// TwinCAT 3 PLC project plc_lfe_vac_fs
// ProgramVersion: 3.1.4022.7
// libraries:
//   L2SI Vacuum Library, * (SLAC)
//   LCLS General, * (SLAC)
//   PMPS, * (SLAC - LCLS)
//   Tc2_Standard, * (Beckhoff Automation GmbH)
//   Tc2_System, * (Beckhoff Automation GmbH)
//   Tc3_Module, * (Beckhoff Automation GmbH)
// project tree:
//   GVLs/ GVL_FS_Devices.TcGVL (not stored)
//   / PlcTask.TcTTO
//   POUs/ MAIN_FS.TcPOU
// (motion and I/O tree: see PLC project plc_lfe_vac)
// real-time tasks:
//   TASK PlcTask: cycle T#10ms, priority 20, ADS port 350
// variable links:
//   plc_lfe_vac/plc_lfe_vac Instance <-> plc_lfe_vac_fs/plc_lfe_vac_fs Instance
//     PlcTask Inputs/GVL_Devices.PA1L0_VFS_01.i_xTrigger <-> PlcTask Outputs/GVL_FS_Devices.PA1L0_VFS_01.q_xTrigger
//     PlcTask Inputs/GVL_Devices.PA1L0_VFS_01.i_xVAC_FAULT_OK <-> PlcTask Outputs/GVL_FS_Devices.PA1L0_VFS_01.q_xVAC_FAULT_OK
//     PlcTask Inputs/GVL_Devices.PA1L0_VFS_01.i_xVFS_Closed <-> PlcTask Outputs/GVL_FS_Devices.PA1L0_VFS_01.q_xVFS_Closed
//     PlcTask Inputs/GVL_Devices.PA1L0_VFS_01.i_xVFS_Open <-> PlcTask Outputs/GVL_FS_Devices.PA1L0_VFS_01.q_xVFS_Open
//     PlcTask Inputs/GVL_Devices.TV3L0_VFS_01_Interface.i_xTrigger <-> PlcTask Outputs/GVL_FS_Devices.TV3L0_VFS_01.q_xTrigger
//     PlcTask Inputs/GVL_Devices.TV3L0_VFS_01_Interface.i_xVAC_FAULT_OK <-> PlcTask Outputs/GVL_FS_Devices.TV3L0_VFS_01.q_xVAC_FAULT_OK
//     PlcTask Inputs/GVL_Devices.TV3L0_VFS_01_Interface.i_xVFS_Closed <-> PlcTask Outputs/GVL_FS_Devices.TV3L0_VFS_01.q_xVFS_Closed
//     PlcTask Inputs/GVL_Devices.TV3L0_VFS_01_Interface.i_xVFS_Open <-> PlcTask Outputs/GVL_FS_Devices.TV3L0_VFS_01.q_xVFS_Open
//     PlcTask Outputs/GVL_Devices.PA1L0_VFS_01.q_xPRESS_OK <-> PlcTask Inputs/GVL_FS_Devices.PA1L0_VFS_01.i_xPress_OK
//     PlcTask Outputs/GVL_Devices.PA1L0_VFS_01.q_xVAC_FAULT_Reset <-> PlcTask Inputs/GVL_FS_Devices.PA1L0_VFS_01.i_xResetFault
//     PlcTask Outputs/GVL_Devices.TV3L0_VFS_01_Interface.q_xPRESS_OK <-> PlcTask Inputs/GVL_FS_Devices.TV3L0_VFS_01.i_xPress_OK
//     PlcTask Outputs/GVL_Devices.TV3L0_VFS_01_Interface.q_xVAC_FAULT_Reset <-> PlcTask Inputs/GVL_FS_Devices.TV3L0_VFS_01.i_xResetFault

CONFIGURATION plc_lfe_vac_fs
    RESOURCE PLC ON TwinCAT3
        TASK PlcTask(INTERVAL := T#10ms, PRIORITY := 20);
        PROGRAM MAIN_FS WITH PlcTask : MAIN_FS;
    END_RESOURCE
END_CONFIGURATION

// ---- POUs/MAIN_FS.TcPOU
PROGRAM MAIN_FS
VAR
	i_xFFReset: INT;
END_VAR

PA1L0_VFS_01(
	i_xPMPS_OK:= TRUE, 
	i_xExt_OK:= TRUE, 
	i_xOverrideMode:= FALSE, 
	iq_stValve=> );
	
TV3L0_VFS_01(
	i_xPMPS_OK:= TRUE, 
	i_xExt_OK:= TRUE, 
	i_xOverrideMode:= FALSE, 
	iq_stValve=> );

END_PROGRAM
